// TIA Portal V16 export
// export: Created 2024-09-05T17:40:14.3876841Z, ExportSetting WithDefaults, DisplayName Totally Integrated Automation Portal, DisplayVersion V16 Update 6, DisplayName TIA Portal Version Control Interface, DisplayVersion V16 Update 2, DisplayName TIA Portal Openness, DisplayVersion V16 Update 6, DisplayName STEP 7 Professional, DisplayVersion V16 Update 6, DisplayName STEP 7 Safety, DisplayVersion V16, DisplayName WinCC Advanced, DisplayVersion V16 Update 6
TYPE "UDT_Servo"
// stored: IsFailsafeCompliant false
   STRUCT
      ModePos : Int;
      EnableAxis : Bool;
      CancelTraversing : Bool;
      IntermediateStop : Bool;
      Positive : Bool;
      Negative : Bool;
      Jog1 : Bool;
      Jog2 : Bool;
      FlyRef : Bool;
      AckError : Bool;
      ExecuteMode : Bool;
      Position : DInt;
      Velocity : DInt;
      OverV : Int;
      OverAcc : Int;
      OverDec : Int;
      AxisEnabled : Bool;
      AxisPosOk : Bool;
      AxisSpFixed : Bool;
      AxisRef : Bool;
      AxisWarn : Bool;
      AxisError : Bool;
      Lockout : Bool;
      ActVelocity : DInt;
      ActPosition : DInt;
      ActMode : Int;
      EPosZSW1 : Word;
      EPosZSW2 : Word;
      ActWarn : Word;
      ActFault : Word;
      Error : Bool;
      Status : Word;
      DiagID : Word;
      data : Struct
         zones : Struct
            inST3jig : Bool;
            inOKpos : Bool;
            inNOKpos : Bool;
            outOfST3zone : Bool;
            outOfOKposZone : Bool;
         END_STRUCT;
      END_STRUCT;
   END_STRUCT;
END_TYPE
